Yaskawa INFORM job: BATMAN_ALL2.JBI

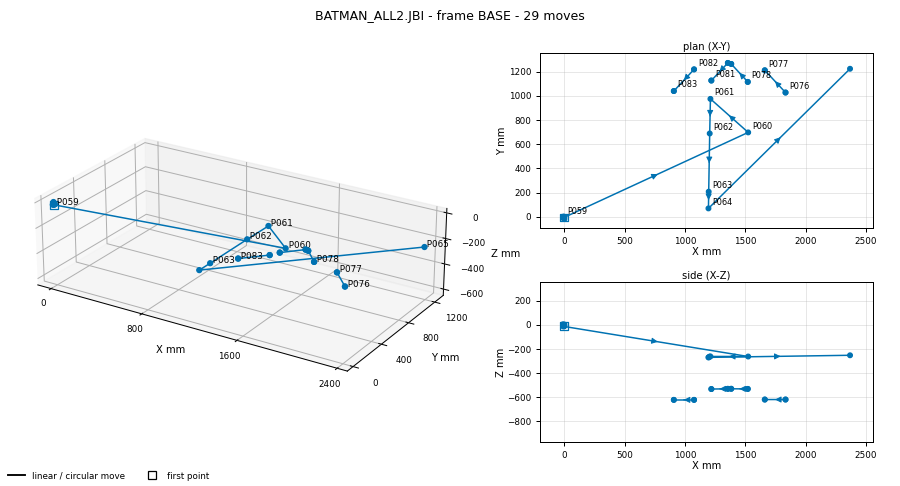
[picture p0: tool path of BATMAN_ALL2.JBI in frame BASE, 29 of 157 moves have a stored position in this frame; points joined in program order, loops and branches not executed]
/JOB
//NAME BATMAN_ALL2
///FOLDERNAME KRIS-SCIANA
//POS
///NPOS 86,86,0,38,0,0
///TOOL 0
///POSTYPE PULSE
///PULSE
C00000=-110506,-37126,-48116,2930,88344,21325
C00001=-114892,-14121,-27107,10658,89628,4728
C00002=-113309,1224,-10446,10482,87095,5056
C00003=-113309,1246,-10200,10482,86959,5045
C00004=-113309,1335,-9328,10485,86476,5004
C00005=-110003,-19046,-27841,10106,86960,6175
C00006=-100624,-28336,-32474,8962,83957,9152
C00007=-100624,-28241,-31795,8967,83593,9126
C00008=-88503,-49798,-46178,7318,80163,13069
C00009=-87519,-47800,-43847,7179,79668,13380
C00010=-87519,-47565,-42796,7191,79148,13350
C00011=-74941,-63128,-53051,5255,76497,17580
C00012=-74079,-59441,-50151,5112,76549,17881
C00013=-74079,-59310,-49676,5116,76325,17872
C00014=-55396,-71634,-57775,1919,74158,24329
C00015=-59223,-66228,-53891,2593,74654,23001
C00016=-59223,-66034,-53265,2596,74369,22996
C00017=-53352,-66899,-53628,1554,73996,25043
C00018=-53352,-66734,-53115,1555,73765,25040
C00019=-64180,-88876,-77181,3423,77531,21350
C00020=-105889,-74463,-75515,8022,88772,8019
C00021=-101467,-10081,-24797,-4145,88218,38060
C00022=-102269,9064,-4514,-5038,90972,37643
C00023=-102269,9132,-3736,-5037,90532,37660
C00024=-106927,-8324,-21894,-4743,92448,36011
C00025=-117713,-25511,-32035,-3960,89286,32487
C00026=-117713,-25417,-31198,-3960,88820,32502
C00027=-121342,-13424,-41304,-3779,101006,30914
C00028=-122365,-2960,-28899,-7414,101341,21577
C00029=-123834,-176,-23705,-7295,99458,21194
C00030=-123834,-264,-23073,-7285,99029,21219
C00031=-125992,-4632,-27757,-7199,99476,20462
C00032=-126961,-4563,-26969,-7139,98946,20168
C00033=-126961,-4621,-26524,-7131,98643,20185
C00034=-128213,-7364,-31817,-7115,100372,19664
C00035=-136462,-13120,-34180,-331,94973,-6688
C00036=-136057,-12661,-33441,-372,94758,-6553
C00037=-136057,-12710,-33041,-372,94486,-6553
C00038=-138935,-4821,-27508,-77,95130,-7505
C00039=-138935,-4905,-26884,-77,94703,-7505
C00040=-154016,-23915,-46161,1473,96922,-12469
C00041=-151429,-25044,-32449,1194,87862,-11704
C00042=-149832,-22551,-30544,1034,87950,-11164
C00043=-149832,-22447,-29458,1034,87335,-11169
C00044=-151805,-19961,-29387,1234,88598,-11822
C00045=-159760,14255,-3469,2028,90388,-14465
C00046=-159397,21628,6319,1975,88147,-14379
C00047=-159397,21727,7358,1975,87559,-14387
C00048=-160803,15292,-4512,2118,91591,-14794
C00049=-147549,18878,-8071,-12007,89530,52437
C00050=-149003,25940,3333,-11752,86001,52284
C00051=-149003,25920,4215,-11756,85457,52336
C00052=-149909,22651,-906,-11580,86775,51906
C00053=-149909,22568,999,-11590,85582,52016
C00054=-149647,22385,-1339,-11629,86944,51982
C00055=-163238,971,-18919,-8991,85058,47564
C00056=-163238,922,-17924,-8996,84429,47610
C00057=-163238,985,-19141,-8988,85202,47554
C00058=-174499,-8933,-26981,-6597,83863,43867
C00059=-174499,-8957,-26535,-6600,83579,43882
C00060=-175724,-10941,-28553,-6329,83702,43466
C00061=-185618,-13902,-30556,-4104,82786,40195
C00062=-185618,-13929,-29820,-4108,82320,40210
C00063=-192158,-22008,-38507,-2587,83246,38002
C00064=-197801,-16314,-31869,-1269,81955,36143
C00065=-197801,-16322,-31570,-1269,81767,36145
C00066=-201132,-17617,-33321,-484,82142,35029
C00067=-201132,-17631,-32925,-484,81891,35030
C00068=-201561,-18787,-38740,-381,84875,34878
C00069=-152433,-2554,-35088,-11190,94372,50378
C00070=-149909,22651,-906,-11580,86775,51906
C00071=-199891,-24598,-44310,-806,86288,35414
C00072=-201584,-39961,-51006,8749,83654,21469
C00073=-110806,-27953,-37591,9544,87699,14562
C00074=-113894,877,-19699,10580,93107,5364
C00075=-72814,-66647,-62566,13351,90363,-8404
C00076=-115805,-17802,-36663,12994,96729,13259
C00077=-115343,1032,-15715,12871,93521,13079
C00078=-116927,-26066,-45887,-4077,97544,32489
C00079=-123423,-3727,-30369,-7384,101759,21178
C00080=-132585,-17564,-40521,-2298,96899,-356
C00081=-153638,2626,-22934,14250,104988,1107
C00082=-149417,-20551,-35648,979,92114,-10995
C00083=-160973,15541,-15915,2153,98738,-14727
C00084=-166397,-29977,-54362,13097,104995,-16051
C00085=-18207,-66647,-62566,13351,90363,-8404
BC00000=234633,5047,784222
BC00001=255264,5047,678683
BC00002=255264,5048,678680
BC00003=255264,5048,678680
BC00004=255264,5048,678680
BC00005=255264,5048,678680
BC00006=255264,5048,678678
BC00007=255264,5048,678678
BC00008=255264,5048,678678
BC00009=255264,5048,678678
BC00010=255264,5048,678678
BC00011=255264,5048,678678
BC00012=255264,5048,678678
BC00013=255264,5048,678678
BC00014=255264,5048,678678
BC00015=255264,5048,678678
BC00016=255264,5048,678678
BC00017=255264,5048,678678
BC00018=255264,5048,678678
BC00019=255264,5048,678678
BC00020=255264,5048,678678
BC00021=255264,5048,678678
BC00022=255264,5048,678678
BC00023=255264,5048,678678
BC00024=255264,5048,678678
BC00025=255264,5048,678678
BC00026=255264,5048,678678
BC00027=255264,5048,678678
BC00028=255264,5048,678678
BC00029=255264,5048,678678
BC00030=255264,5048,678678
BC00031=255264,5048,678678
BC00032=255264,5048,678678
BC00033=255264,5048,678678
BC00034=255264,5048,678678
BC00035=255264,5048,678678
BC00036=255264,5048,678678
BC00037=255264,5048,678678
BC00038=255264,5048,678678
BC00039=255264,5048,678678
BC00040=255264,5048,678678
BC00041=255264,5048,678678
BC00042=255264,5048,678678
BC00043=255264,5048,678678
BC00044=255264,5048,678678
BC00045=255264,5048,678678
BC00046=255263,5049,678675
BC00047=255263,5049,678675
BC00048=255263,5049,678675
BC00049=255264,5046,617469
BC00050=255264,5046,617469
BC00051=255264,5046,617469
BC00052=255264,5046,617469
BC00053=255264,5046,617469
BC00054=255264,5046,617469
BC00055=255264,5046,617469
BC00056=255264,5046,617469
BC00057=255264,5046,617469
BC00058=255264,5046,617469
BC00059=255264,5046,617469
BC00060=255264,5046,617469
BC00061=255264,5046,617469
BC00062=255264,5046,617469
BC00063=255264,5046,617469
BC00064=255264,5046,617469
BC00065=255264,5046,617469
BC00066=255264,5046,617469
BC00067=255264,5046,617469
BC00068=255264,5046,617469
BC00069=255264,5047,617466
BC00070=255264,5046,617469
BC00071=255264,5046,617469
BC00072=255264,5047,821128
BC00073=255264,5047,760053
BC00074=255264,5048,678680
BC00075=255264,5048,678680
BC00076=255264,5048,678680
BC00077=255264,5048,678680
BC00078=255264,5048,678680
BC00079=255264,5048,678680
BC00080=255264,5048,678680
BC00081=255264,5048,678680
BC00082=255264,5048,678680
BC00083=255264,5048,678680
BC00084=255264,5048,678680
BC00085=143206,5048,998327
///POSTYPE BASE
///RECTAN
///RCONF 0,0,0,0,0,0,0,0,0,0,0,0,0,0,0,0,0,0,0,0,0,0,0,0
P00059=-2.448,-6.714,-12.718,0.0000,0.0000,0.0000
P00060=1524.284,698.404,-261.973,-0.4635,36.8346,-1.2388
P00061=1211.499,975.999,-261.374,0.5148,35.2356,175.5099
P00062=1205.574,689.500,-262.704,0.5159,35.2461,175.5270
P00063=1197.217,207.358,-268.729,0.4863,35.2395,175.4586
P00064=1195.199,68.975,-269.171,0.5092,35.2366,175.4908
P00065=2367.684,1225.356,-251.745,0.6375,35.5356,-175.5535
P00070=2.449,-18.318,2.615,0.0000,0.0000,0.0000
P00071=-2.048,-0.034,-9.092,0.0000,0.0000,0.0000
P00072=-1.595,-0.049,-6.373,0.0000,0.0000,0.0000
P00073=-8.474,-10.331,-11.894,0.0000,0.0000,0.0000
P00074=1.731,-3.007,-10.460,0.0000,0.0000,0.0000
///RCONF 0,1,0,0,0,0,0,0,0,0,0,0,0,0,0,0,0,0,0,0,0,0,0,0
P00075=-9.634,0.014,4.922,0.0000,0.0000,0.0000
///RCONF 0,0,0,0,0,0,0,0,0,0,0,0,0,0,0,0,0,0,0,0,0,0,0,0
P00076=1833.500,1028.615,-618.215,10.0256,37.5190,56.2681
P00077=1661.766,1212.555,-618.325,10.0309,37.5577,56.2858
P00078=1520.740,1116.757,-530.271,10.0398,37.5578,56.2925
P00079=1383.754,1265.334,-529.217,10.0293,37.5461,56.2787
P00080=1355.833,1273.708,-529.583,10.0283,37.5305,126.4716
P00081=1219.184,1127.874,-531.327,10.0137,37.5345,126.4324
P00082=1075.995,1220.294,-620.895,10.0203,37.5289,126.4576
P00083=908.434,1040.970,-620.895,10.0141,37.5419,126.4584
P00098=-1.000,0.000,-2.000,0.0000,0.0000,-60.0000
P00099=-10.497,4.418,3.734,0.0000,0.0000,0.0000
P00105=-13.000,6.000,-2.500,0.0000,0.0000,0.0000
P00106=13.000,-13.000,-3.000,0.0000,0.0000,0.0000
P00107=-12.000,8.000,-3.000,0.0000,0.0000,0.0000
P00108=0.000,0.000,-3.000,0.0000,0.0000,0.0000
P00110=13.000,10.000,-3.000,0.0000,0.0000,0.0000
P00111=-15.000,-15.000,-2.000,0.0000,0.0000,0.0000
P00112=15.000,7.000,-2.500,0.0000,0.0000,0.0000
P00113=-8.000,-10.000,-3.000,0.0000,0.0000,0.0000
P00114=10.000,-8.000,-3.000,0.0000,0.0000,0.0000
P00124=0.000,50.000,0.000,0.0000,0.0000,0.0000
P00125=0.000,0.000,2.400,0.0000,0.0000,0.0000
P00126=-50.000,0.000,0.000,0.0000,0.0000,0.0000
P00127=50.000,0.000,0.000,0.0000,0.0000,0.0000
P00170=4.000,4.000,-1.000,-10.0000,10.0000,-30.0000
P00171=-8.000,11.000,-2.000,0.0000,0.0000,-60.0000
//INST
///DATE 2024/07/30 17:33
///COMM NOWY SEARCH
///ATTR SC,RW
///GROUP1 RB1,BS1
NOP
SFTOF
CALL JOB:ONLYCUT-R1_LONG
MOVJ C00000 BC00000 VJ=15.00
MOVJ C00001 BC00001 VJ=15.00
'POMIAR PRAWA STRONA
MOVL C00002 BC00002 V=250.0
'1
MOVL C00003 BC00003 V=166.7
MOVL C00004 BC00004 V=16.7 PL=0 SRCH RIN#(1)=ON T=1.00 DIS=20.0
TIMER T=0.20
IMOV P125 V=13.3 PL=0
TIMER T=0.20
IMOV P127 V=13.3 PL=0 SRCH RIN#(1)=ON DIS=20.0
TIMER T=0.20
GETS PX070 $PX001
TIMER T=0.10
MOVJ C00005 BC00005 VJ=15.00
'2
MOVL C00006 BC00006 V=50.0
MOVL C00007 BC00007 V=16.7 PL=0 SRCH RIN#(1)=ON T=1.00 DIS=20.0
TIMER T=0.20
IMOV P125 V=13.3 PL=0
TIMER T=0.20
IMOV P127 V=13.3 PL=0 SRCH RIN#(1)=ON DIS=20.0
TIMER T=0.20
GETS PX071 $PX001
TIMER T=0.10
MOVJ C00008 BC00008 VJ=15.00
'3
MOVL C00009 BC00009 V=50.0
MOVL C00010 BC00010 V=16.7 PL=0 SRCH RIN#(1)=ON T=1.00 DIS=20.0
TIMER T=0.20
IMOV P125 V=13.3 PL=0
TIMER T=0.20
IMOV P127 V=13.3 PL=0 SRCH RIN#(1)=ON DIS=20.0
TIMER T=0.20
GETS PX072 $PX001
TIMER T=0.10
MOVJ C00011 BC00011 VJ=15.00
'4
MOVL C00012 BC00012 V=50.0
MOVL C00013 BC00013 V=16.7 PL=0 SRCH RIN#(1)=ON T=1.00 DIS=20.0
TIMER T=0.20
IMOV P125 V=13.3 PL=0
TIMER T=0.20
IMOV P127 V=13.3 PL=0 SRCH RIN#(1)=ON DIS=20.0
TIMER T=0.20
GETS PX073 $PX001
TIMER T=0.10
MOVJ C00014 BC00014 VJ=15.00
'5
MOVL C00015 BC00015 V=50.0
MOVL C00016 BC00016 V=16.7 PL=0 SRCH RIN#(1)=ON T=1.00 DIS=20.0
TIMER T=0.20
IMOV P125 V=13.3 PL=0
TIMER T=0.20
IMOV P127 V=13.3 PL=0 SRCH RIN#(1)=ON DIS=20.0
TIMER T=0.20
GETS PX074 $PX001
TIMER T=0.10
MOVL C00017 BC00017 V=50.0
MOVL C00018 BC00018 V=16.7 PL=0 SRCH RIN#(1)=ON T=1.00 DIS=20.0
TIMER T=0.20
IMOV P125 V=13.3 PL=0
TIMER T=0.20
IMOV P127 V=13.3 PL=0 SRCH RIN#(1)=ON DIS=20.0
TIMER T=0.20
GETS PX075 $PX001
TIMER T=0.10
MOVJ C00019 BC00019 VJ=15.00
MOVJ C00020 BC00020 VJ=30.00
'POMIAR BATMAN
MOVJ C00021 BC00021 VJ=30.00
MOVL C00022 BC00022 V=166.7
MOVL C00023 BC00023 V=13.3 PL=0 SRCH RIN#(1)=ON T=1.00 DIS=20.0
TIMER T=0.20
IMOV P125 V=13.3 PL=0
TIMER T=0.20
IMOV P124 V=13.3 PL=0 SRCH RIN#(1)=ON DIS=20.0
TIMER T=0.20
GETS PX076 $PX001
TIMER T=0.10
MOVJ C00024 BC00024 VJ=30.00
MOVL C00025 BC00025 V=166.7
MOVL C00026 BC00026 V=16.7 PL=0 SRCH RIN#(1)=ON T=1.00 DIS=20.0
TIMER T=0.20
IMOV P125 V=13.3 PL=0
TIMER T=0.20
IMOV P124 V=13.3 PL=0 SRCH RIN#(1)=ON DIS=20.0
TIMER T=0.20
GETS PX077 $PX001
TIMER T=0.10
MOVJ C00027 BC00027 VJ=30.00
MOVJ C00028 BC00028 VJ=30.00
MOVL C00029 BC00029 V=166.7
MOVL C00030 BC00030 V=16.7 PL=0 SRCH RIN#(1)=ON T=1.00 DIS=20.0
TIMER T=0.20
IMOV P125 V=13.3 PL=0
TIMER T=0.20
IMOV P124 V=13.3 PL=0 SRCH RIN#(1)=ON DIS=20.0
TIMER T=0.20
GETS PX078 $PX001
TIMER T=0.10
MOVJ C00031 BC00031 VJ=30.00
MOVL C00032 BC00032 V=166.7
MOVL C00033 BC00033 V=16.7 PL=0 SRCH RIN#(1)=ON T=1.00 DIS=20.0
TIMER T=0.20
IMOV P125 V=13.3 PL=0
TIMER T=0.20
IMOV P124 V=13.3 PL=0 SRCH RIN#(1)=ON DIS=20.0
TIMER T=0.20
GETS PX079 $PX001
TIMER T=0.10
MOVJ C00034 BC00034 VJ=30.00
MOVJ C00035 BC00035 VJ=30.00
MOVL C00036 BC00036 V=166.7
MOVL C00037 BC00037 V=16.7 PL=0 SRCH RIN#(1)=ON T=1.00 DIS=20.0
TIMER T=0.20
IMOV P125 V=13.3 PL=0
TIMER T=0.20
IMOV P124 V=13.3 PL=0 SRCH RIN#(1)=ON DIS=20.0
TIMER T=0.20
GETS PX080 $PX001
TIMER T=0.10
MOVL C00038 BC00038 V=166.7
MOVL C00039 BC00039 V=16.7 PL=0 SRCH RIN#(1)=ON T=1.00 DIS=20.0
TIMER T=0.20
IMOV P125 V=13.3 PL=0
TIMER T=0.20
IMOV P124 V=13.3 PL=0 SRCH RIN#(1)=ON DIS=20.0
TIMER T=0.20
GETS PX081 $PX001
TIMER T=0.10
MOVJ C00040 BC00040 VJ=30.00
MOVJ C00041 BC00041 VJ=30.00
MOVL C00042 BC00042 V=166.7
MOVL C00043 BC00043 V=16.7 PL=0 SRCH RIN#(1)=ON T=1.00 DIS=20.0
TIMER T=0.20
IMOV P125 V=13.3 PL=0
TIMER T=0.20
IMOV P124 V=13.3 PL=0 SRCH RIN#(1)=ON DIS=20.0
TIMER T=0.20
GETS PX082 $PX001
TIMER T=0.10
MOVJ C00044 BC00044 VJ=15.00
MOVJ C00045 BC00045 VJ=30.00
MOVL C00046 BC00046 V=166.7
MOVL C00047 BC00047 V=16.7 PL=0 SRCH RIN#(1)=ON T=1.00 DIS=20.0
TIMER T=0.20
IMOV P125 V=23.0 PL=0
TIMER T=0.20
IMOV P124 V=23.0 PL=0 SRCH RIN#(1)=ON DIS=20.0
TIMER T=0.20
GETS PX083 $PX001
TIMER T=0.10
MOVJ C00048 BC00048 VJ=30.00
'KONIEC POMIAR BATMAN 1STR
SFTOF
MOVJ C00049 BC00049 VJ=15.00
'1
MOVL C00050 BC00050 V=166.7
MOVL C00051 BC00051 V=16.7 PL=0 SRCH RIN#(1)=ON T=1.00 DIS=20.0
TIMER T=0.20
IMOV P125 V=13.3 PL=0
TIMER T=0.20
IMOV P126 V=13.3 PL=0 SRCH RIN#(1)=ON DIS=20.0
TIMER T=0.20
GETS PX059 $PX001
TIMER T=0.10
MOVL C00052 BC00052 V=166.7
MOVL C00053 BC00053 V=16.7 PL=0 SRCH RIN#(1)=ON T=1.00 DIS=20.0
TIMER T=0.20
IMOV P125 V=13.3 PL=0
TIMER T=0.20
IMOV P126 V=13.3 PL=0 SRCH RIN#(1)=ON DIS=20.0
TIMER T=0.20
GETS PX060 $PX001
TIMER T=0.10
MOVJ C00054 BC00054 VJ=0.78
'2
MOVL C00055 BC00055 V=50.0
MOVL C00056 BC00056 V=16.7 PL=0 SRCH RIN#(1)=ON T=1.00 DIS=20.0
TIMER T=0.20
IMOV P125 V=13.3 PL=0
TIMER T=0.20
IMOV P126 V=13.3 PL=0 SRCH RIN#(1)=ON DIS=20.0
TIMER T=0.20
GETS PX061 $PX001
TIMER T=0.10
MOVJ C00057 BC00057 VJ=0.78
'3
MOVL C00058 BC00058 V=50.0
MOVL C00059 BC00059 V=16.7 PL=0 SRCH RIN#(1)=ON T=1.00 DIS=20.0
TIMER T=0.20
IMOV P125 V=13.3 PL=0
TIMER T=0.20
IMOV P126 V=13.3 PL=0 SRCH RIN#(1)=ON DIS=20.0
TIMER T=0.20
GETS PX062 $PX001
TIMER T=0.10
MOVJ C00060 BC00060 VJ=0.78
'4
MOVL C00061 BC00061 V=50.0
MOVL C00062 BC00062 V=16.7 PL=0 SRCH RIN#(1)=ON T=1.00 DIS=20.0
TIMER T=0.20
IMOV P125 V=13.3 PL=0
TIMER T=0.20
IMOV P126 V=13.3 PL=0 SRCH RIN#(1)=ON DIS=20.0
TIMER T=0.20
GETS PX063 $PX001
TIMER T=0.10
MOVJ C00063 BC00063 VJ=30.00
'5
MOVL C00064 BC00064 V=50.0
MOVL C00065 BC00065 V=16.7 PL=0 SRCH RIN#(1)=ON T=1.00 DIS=20.0
TIMER T=0.20
IMOV P125 V=13.3 PL=0
TIMER T=0.20
IMOV P126 V=13.3 PL=0 SRCH RIN#(1)=ON DIS=20.0
TIMER T=0.20
GETS PX064 $PX001
TIMER T=0.10
MOVL C00066 BC00066 V=50.0
MOVL C00067 BC00067 V=16.7 PL=0 SRCH RIN#(1)=ON T=1.00 DIS=20.0
TIMER T=0.20
IMOV P125 V=13.3 PL=0
TIMER T=0.20
IMOV P126 V=13.3 PL=0 SRCH RIN#(1)=ON DIS=20.0
TIMER T=0.20
GETS PX065 $PX001
TIMER T=0.10
MOVJ C00068 BC00068 VJ=15.00
'********
'********
'********
MOVJ C00069 BC00069 VJ=15.00
MOVL C00070 BC00070 V=333.3
MACRO1 MJ#(0) ARGF7
SFTOF
SFTON P170
MOVL P059 V=83.3
ARCON
SFTOF
SFTON P099
MOVL P060 V=10.8
MOVL P061 V=10.8
MOVL P062 V=10.8
MOVL P063 V=10.8
MOVL P064 V=10.8
MOVL P065 V=10.8
ARCOF
MOVJ C00071 BC00071 VJ=15.00
SFTOF
MOVJ C00072 BC00072 VJ=15.00
MOVJ C00073 BC00073 VJ=15.00
SFTON P171
MOVJ C00074 BC00074 VJ=15.00
MOVL P070 V=83.3
ARCON
SFTOF
SFTON P098
MOVL P071 V=10.8
MOVL P072 V=10.8
MOVL P073 V=10.8
MOVL P074 V=10.8
MOVL P075 V=10.8
ARCOF
SFTOF
MOVJ C00075 BC00075 VJ=15.00
MOVJ C00076 BC00076 VJ=30.00
MOVJ C00077 BC00077 VJ=30.00
SFTON P110
MOVL P076 V=83.3
SFTOF
ARCON
SFTON P108
MOVL P076 V=10.8
MOVL P077 V=10.8
SFTON P111
MOVL P077 V=10.8
ARCOF
SFTOF
MOVJ C00078 BC00078 VJ=30.00
MOVJ C00079 BC00079 VJ=30.00
SFTON P112
MOVL P078 V=83.3
ARCON
SFTOF
SFTON P108
MOVL P078 V=10.8
MOVL P079 V=10.8
SFTOF
SFTON P113
MOVL P079 V=10.8
ARCOF
SFTOF
MOVJ C00080 BC00080 VJ=30.00
SFTON P114
MOVL P080 V=83.3
SFTOF
ARCON
SFTON P108
MOVL P080 V=10.8
MOVL P081 V=10.8
SFTOF
SFTON P105
MOVL P081 V=10.8
SFTOF
ARCOF
MOVJ C00081 BC00081 VJ=30.00
MOVJ C00082 BC00082 VJ=30.00
SFTON P106
MOVL P082 V=83.3
SFTOF
ARCON
SFTON P108
MOVL P082 V=10.8
MOVL P083 V=10.8
SFTOF
SFTON P107
MOVL P083 V=10.8
SFTOF
ARCOF
MOVJ C00083 BC00083 VJ=30.00
MOVJ C00084 BC00084 VJ=30.00
MOVJ C00085 BC00085 VJ=30.00
CALL JOB:ONLYCUT-R1_LONG
END
